PROGRAM Permissives
VAR

	stPermissives			: ST_PermissivesToMainPLC;
	
	AdminFaultBypassOn		: BOOL;
	
	i : INT := 1;
	j : INT := 1;	
END_VAR

//HMI Admin bypass button
AdminFaultBypassOn := HMI_DB.SafetyOK;

//Check to see if any coil is disabled
IF Devices.Coil[1].CoilEnabled = FALSE OR
	Devices.Coil[2].CoilEnabled = FALSE OR
	Devices.Coil[3].CoilEnabled = FALSE OR
	Devices.Coil[4].CoilEnabled = FALSE OR
	Devices.Coil[5].CoilEnabled = FALSE OR
	Devices.Coil[6].CoilEnabled = FALSE OR
	Devices.Coil[7].CoilEnabled = FALSE OR
	Devices.Coil[8].CoilEnabled = FALSE OR
	Devices.Coil[9].CoilEnabled = FALSE OR
	Devices.Coil[10].CoilEnabled = FALSE 
	THEN
		Permissives_DB.AnyCoilDisabled := TRUE;
	ELSE
		Permissives_DB.AnyCoilDisabled := FALSE;
END_IF;

//check to see if each LCP system is ready based on the selected safety parameters.
FOR i := 1 TO 10 BY 1 DO
	IF Devices.Coil[i].AC_Interlock_RlyClose = TRUE AND 
		Devices.Coil[i].ChargeRelay_closed = TRUE AND
		Devices.Coil[i].CoilTemperatureHigh = FALSE AND
		Devices.Coil[i].DumpResistorTemperatureHigh = FALSE AND
		Devices.Coil[i].DumpRelay1_closed = TRUE AND
		Devices.Coil[i].DumpRelay2_closed = TRUE AND
		Devices.Coil[i].FlybackD1_Alive = TRUE AND
		Devices.Coil[i].FlybackD2_Alive = TRUE AND
		Devices.Coil[i].GroundLoopCurrentDetected = FALSE AND
		Devices.Coil[i].Local_StopPB_Pressed = FALSE AND
		Devices.Coil[i].LossPneumaticPressure = FALSE 
		THEN
			Devices.Coil[i].SystemReady := TRUE;
		ELSE
			Devices.Coil[i].SystemReady := FALSE;
	END_IF;
END_FOR;


//Safety Permissives
	//Interlock Safety
	IF (Devices.Coil[1].AC_Interlock_RlyClose = TRUE OR Devices.Coil[1].CoilEnabled = FALSE) AND 
		(Devices.Coil[2].AC_Interlock_RlyClose = TRUE OR Devices.Coil[2].CoilEnabled = FALSE) AND 
		(Devices.Coil[3].AC_Interlock_RlyClose = TRUE OR Devices.Coil[3].CoilEnabled = FALSE) AND
		(Devices.Coil[4].AC_Interlock_RlyClose = TRUE OR Devices.Coil[4].CoilEnabled = FALSE) AND
		(Devices.Coil[5].AC_Interlock_RlyClose = TRUE OR Devices.Coil[5].CoilEnabled = FALSE) AND
		(Devices.Coil[6].AC_Interlock_RlyClose = TRUE OR Devices.Coil[6].CoilEnabled = FALSE) AND
		(Devices.Coil[7].AC_Interlock_RlyClose = TRUE OR Devices.Coil[7].CoilEnabled = FALSE) AND
		(Devices.Coil[8].AC_Interlock_RlyClose = TRUE OR Devices.Coil[8].CoilEnabled = FALSE) AND
		(Devices.Coil[9].AC_Interlock_RlyClose = TRUE OR Devices.Coil[9].CoilEnabled = FALSE) AND 
		(Devices.Coil[10].AC_Interlock_RlyClose = TRUE OR Devices.Coil[10].CoilEnabled = FALSE)
		
		THEN 
			Permissives_DB.AllacInterlock_Closed := TRUE;
		ELSE 
			Permissives_DB.AllacInterlock_Closed := FALSE;
	END_IF;

	//Coil Temperature
	IF Devices.Coil[1].CoilTemperatureHigh = FALSE AND
		Devices.Coil[2].CoilTemperatureHigh = FALSE 
		THEN
			Permissives_DB.All_Coil_TemperatureOK := TRUE;
		ELSE 
			Permissives_DB.All_Coil_TemperatureOK := FALSE;
	END_IF;

	//Dump Resistor Temperature
	IF Devices.Coil[1].DumpResistorTemperatureHigh = FALSE AND
		Devices.Coil[2].DumpResistorTemperatureHigh = FALSE 
		THEN
			Permissives_DB.AllDumpResistorTempOK := TRUE;
		ELSE 
			Permissives_DB.AllDumpResistorTempOK := FALSE;
	END_IF;
	
	//Ground loop current
	IF Devices.Coil[1].GroundLoopCurrentDetected = FALSE AND
		Devices.Coil[2].GroundLoopCurrentDetected = FALSE 
		THEN
			Permissives_DB.NoGroundLoopCurrentDetected := TRUE;
		ELSE 
			Permissives_DB.NoGroundLoopCurrentDetected := FALSE;
	END_IF;
	
	//Flyback Diodes - Not enought time for PI3 - temporarily disabled for PI3
(*	IF ((Devices.coil[1].FlybackD1_Alive = TRUE AND Devices.coil[1].FlybackD2_Alive = TRUE) OR Devices.Coil[1].CoilEnabled = FALSE) AND
		((Devices.coil[2].FlybackD1_Alive = TRUE AND Devices.coil[2].FlybackD2_Alive = TRUE) OR Devices.Coil[2].CoilEnabled = FALSE)
		THEN 
			AllFlybackDiodes_Alive := TRUE;
		ELSE 
			AllFlybackDiodes_Alive := FALSE;
	END_IF;
*)	
	IF (Permissives_DB.All_Coil_TemperatureOK = TRUE AND
		Permissives_DB.AllDumpResistorTempOK = TRUE AND
		Permissives_DB.NoGroundLoopCurrentDetected = TRUE AND
		//AllFlybackDiodes_Alive = TRUE AND 
		Trips_DB.AnyACInterlockFail = FALSE AND
		Trips_DB.AnyHVisoRelayFailed = FALSE AND
		Trips_DB.AnyChargeRlyFail = FALSE AND
		Trips_DB.AnyDumpRlyFail = FALSE AND
		Trips_DB.AnyEstopPressed = FALSE AND
		Permissives_DB.AlldcPSUok = TRUE AND
		MCP_IO.CageEstopCircuitOK = TRUE) OR HMI_DB.SafetyOK = TRUE 
		THEN
			Permissives_DB.SafetyOK := TRUE;
		ELSE 
			Permissives_DB.SafetyOK := FALSE; 
	END_IF;

//Charger Active Status - obsolete
(*
IF (Devices.Coil[1].PSU0_active = TRUE OR Devices.Coil[1].CoilEnabled = FALSE) AND
	(Devices.Coil[2].PSU0_active = TRUE OR Devices.Coil[2].CoilEnabled = FALSE) //AND
	//Coil3.PSU.active AND 
	THEN 
		AllChargers_Active := TRUE;
	ELSE 
		AllChargers_Active := FALSE;
END_IF;
*)

IF (Devices.Coil[1].PSU1_DCOK = TRUE OR Devices.Coil[1].CoilEnabled = FALSE) AND
	(Devices.Coil[2].PSU1_DCOK = TRUE OR Devices.Coil[2].CoilEnabled = FALSE) (*AND Coil3.PSU.active*) AND
	MCP_IO.PSU1_DCOK = TRUE
	THEN 
		Permissives_DB.AlldcPSUok := TRUE;
	ELSE 
		Permissives_DB.AlldcPSUok := FALSE;
END_IF;

//Charger Enabled Status
IF (Devices.Coil[1].ChargerIsEnabled = TRUE OR Devices.Coil[1].CoilEnabled = FALSE) AND
	(Devices.Coil[2].ChargerIsEnabled = TRUE OR Devices.Coil[2].CoilEnabled = FALSE) AND
	(Devices.Coil[3].ChargerIsEnabled = TRUE OR Devices.Coil[3].CoilEnabled = FALSE) AND
	(Devices.Coil[4].ChargerIsEnabled = TRUE OR Devices.Coil[4].CoilEnabled = FALSE) AND
	(Devices.Coil[5].ChargerIsEnabled = TRUE OR Devices.Coil[5].CoilEnabled = FALSE) AND
	(Devices.Coil[6].ChargerIsEnabled = TRUE OR Devices.Coil[6].CoilEnabled = FALSE) AND
	(Devices.Coil[7].ChargerIsEnabled = TRUE OR Devices.Coil[7].CoilEnabled = FALSE) AND	
	(Devices.Coil[8].ChargerIsEnabled = TRUE OR Devices.Coil[8].CoilEnabled = FALSE) AND
	(Devices.Coil[9].ChargerIsEnabled = TRUE OR Devices.Coil[9].CoilEnabled = FALSE) AND
	(Devices.Coil[10].ChargerIsEnabled = TRUE OR Devices.Coil[10].CoilEnabled = FALSE) 
	THEN 
		Permissives_DB.AllChargerEnabled := TRUE;
	ELSE 
		Permissives_DB.AllChargerEnabled := FALSE;
END_IF

//???? need more work
IF ((Devices.Coil[1].chargerSetpoint >= Setpoints.Coil[1].RecipeLocal.chargerSetpoint) OR Devices.Coil[1].CoilEnabled = FALSE) AND
	((Devices.Coil[2].chargerSetpoint >= Setpoints.Coil[2].RecipeLocal.chargerSetpoint) OR Devices.Coil[2].CoilEnabled = FALSE) AND 
	((Devices.Coil[3].chargerSetpoint >= Setpoints.Coil[3].RecipeLocal.chargerSetpoint) OR Devices.Coil[3].CoilEnabled = FALSE) AND
	((Devices.Coil[4].chargerSetpoint >= Setpoints.Coil[4].RecipeLocal.chargerSetpoint) OR Devices.Coil[4].CoilEnabled = FALSE) AND
	((Devices.Coil[5].chargerSetpoint >= Setpoints.Coil[5].RecipeLocal.chargerSetpoint) OR Devices.Coil[5].CoilEnabled = FALSE) AND
	((Devices.Coil[6].chargerSetpoint >= Setpoints.Coil[6].RecipeLocal.chargerSetpoint) OR Devices.Coil[6].CoilEnabled = FALSE) AND
	((Devices.Coil[7].chargerSetpoint >= Setpoints.Coil[7].RecipeLocal.chargerSetpoint) OR Devices.Coil[7].CoilEnabled = FALSE) AND
	((Devices.Coil[8].chargerSetpoint >= Setpoints.Coil[8].RecipeLocal.chargerSetpoint) OR Devices.Coil[8].CoilEnabled = FALSE) AND
	((Devices.Coil[9].chargerSetpoint >= Setpoints.Coil[9].RecipeLocal.chargerSetpoint) OR Devices.Coil[9].CoilEnabled = FALSE) AND
	((Devices.Coil[10].chargerSetpoint >= Setpoints.Coil[10].RecipeLocal.chargerSetpoint) OR Devices.Coil[10].CoilEnabled = FALSE)
	THEN
		GVL.AllChargerReadywithSP := TRUE;
	ELSE
		GVL.AllChargerReadywithSP := FALSE;
END_IF;

//check to see if all cap voltage ready to shoot
FOR i := 1 TO 10 BY 1 DO
		IF ((Devices.Coil[i].CapVoltage[1] >= Devices.Coil[i].chargerSetpoint) AND
			(Devices.Coil[i].CapVoltage[2] >= Devices.Coil[i].chargerSetpoint) AND
			(Devices.Coil[i].CapVoltage[3] >= Devices.Coil[i].chargerSetpoint) AND
			(Devices.Coil[i].CapVoltage[4] >= Devices.Coil[i].chargerSetpoint) AND
			(Devices.Coil[i].CapVoltage[5] >= Devices.Coil[i].chargerSetpoint) AND
			(Devices.Coil[i].CapVoltage[6] >= Devices.Coil[i].chargerSetpoint) AND
			(Devices.Coil[i].CapVoltage[7] >= Devices.Coil[i].chargerSetpoint) AND
			(Devices.Coil[i].CapVoltage[8] >= Devices.Coil[i].chargerSetpoint) AND
			(Devices.Coil[i].CapVoltage[9] >= Devices.Coil[i].chargerSetpoint) AND
			(Devices.Coil[i].CapVoltage[10] >= Devices.Coil[i].chargerSetpoint)) OR 
			Devices.Coil[i].CoilEnabled = FALSE
		THEN
			Devices.Coil[i].AllCapsCharged := TRUE;
	END_IF
END_FOR;
//check to see if all coils are charged
IF Devices.Coil[1].AllCapsCharged = TRUE AND 
	Devices.Coil[2].AllCapsCharged = TRUE AND 
	Devices.Coil[3].AllCapsCharged = TRUE AND 
	Devices.Coil[4].AllCapsCharged = TRUE AND 
	Devices.Coil[5].AllCapsCharged = TRUE AND 
	Devices.Coil[6].AllCapsCharged = TRUE AND 
	Devices.Coil[7].AllCapsCharged = TRUE AND 
	Devices.Coil[8].AllCapsCharged = TRUE AND 
	Devices.Coil[9].AllCapsCharged = TRUE AND 
	Devices.Coil[10].AllCapsCharged = TRUE 
THEN 
	Permissives_DB.AllCoilCapsCharged := TRUE;
ELSE
	Permissives_DB.AllCoilCapsCharged := FALSE;	
END_IF

//check to see if all cap voltage drops to 1
IF ((Devices.Coil[i].CapVoltage[1] <= 1) AND
	(Devices.Coil[i].CapVoltage[2] <= 1) AND
	(Devices.Coil[i].CapVoltage[3] <= 1) AND
	(Devices.Coil[i].CapVoltage[4] <= 1) AND
	(Devices.Coil[i].CapVoltage[5] <= 1) AND
	(Devices.Coil[i].CapVoltage[6] <= 1) AND
	(Devices.Coil[i].CapVoltage[7] <= 1) AND
	(Devices.Coil[i].CapVoltage[8] <= 1) AND
	(Devices.Coil[i].CapVoltage[9] <= 1) AND
	(Devices.Coil[i].CapVoltage[10] <= 1)) OR 
	Devices.Coil[i].CoilEnabled = FALSE
THEN
	Devices.Coil[i].AllCapsCharged := FALSE;
END_IF;



//Charger Relay
IF Devices.Coil[1].ChargeRelay_closed = FALSE AND
	Devices.Coil[2].ChargeRelay_closed = FALSE 
	//coil n
	THEN
		Permissives_DB.AllChargerRelay_Closed := TRUE;
	ELSE 
		Permissives_DB.AllChargerRelay_Closed := FALSE;
END_IF

	
//Dump Relay Status
(* obsolete - use the one at the bottom
IF ((Devices.Coil[1].DumpRelay1_closed = FALSE AND Devices.Coil[1].DumpRelay2_closed = FALSE) OR Devices.Coil[1].CoilEnabled = FALSE) AND
	((Devices.Coil[2].DumpRelay1_closed = FALSE AND Devices.Coil[2].DumpRelay2_closed = FALSE) OR Devices.Coil[2].CoilEnabled = FALSE) AND
	((Devices.Coil[3].DumpRelay1_closed = FALSE AND Devices.Coil[3].DumpRelay2_closed = FALSE) OR Devices.Coil[3].CoilEnabled = FALSE) AND
	((Devices.Coil[4].DumpRelay1_closed = FALSE AND Devices.Coil[4].DumpRelay2_closed = FALSE) OR Devices.Coil[4].CoilEnabled = FALSE) AND
	((Devices.Coil[5].DumpRelay1_closed = FALSE AND Devices.Coil[5].DumpRelay2_closed = FALSE) OR Devices.Coil[5].CoilEnabled = FALSE) AND
	((Devices.Coil[6].DumpRelay1_closed = FALSE AND Devices.Coil[6].DumpRelay2_closed = FALSE) OR Devices.Coil[6].CoilEnabled = FALSE) AND
	((Devices.Coil[7].DumpRelay1_closed = FALSE AND Devices.Coil[7].DumpRelay2_closed = FALSE) OR Devices.Coil[7].CoilEnabled = FALSE) AND
	((Devices.Coil[8].DumpRelay1_closed = FALSE AND Devices.Coil[8].DumpRelay2_closed = FALSE) OR Devices.Coil[8].CoilEnabled = FALSE) AND
	((Devices.Coil[9].DumpRelay1_closed = FALSE AND Devices.Coil[9].DumpRelay2_closed = FALSE) OR Devices.Coil[9].CoilEnabled = FALSE) AND
	((Devices.Coil[10].DumpRelay1_closed = FALSE AND Devices.Coil[10].DumpRelay2_closed = FALSE) OR Devices.Coil[10].CoilEnabled = FALSE)

	THEN
		AllDumpRelayOpen := TRUE;
		ELSE 
			AllDumpRelayOpen := FALSE;
END_IF;
*)	
IF ((Devices.Coil[1].DumpRelay1_closed = TRUE AND Devices.Coil[1].DumpRelay2_closed = TRUE) OR Devices.Coil[1].CoilEnabled = FALSE) AND
	((Devices.Coil[2].DumpRelay1_closed = TRUE AND Devices.Coil[2].DumpRelay2_closed = TRUE) OR Devices.Coil[2].CoilEnabled = FALSE) AND
	((Devices.Coil[3].DumpRelay1_closed = TRUE AND Devices.Coil[3].DumpRelay2_closed = TRUE) OR Devices.Coil[3].CoilEnabled = FALSE) AND
	((Devices.Coil[4].DumpRelay1_closed = TRUE AND Devices.Coil[4].DumpRelay2_closed = TRUE) OR Devices.Coil[4].CoilEnabled = FALSE) AND
	((Devices.Coil[5].DumpRelay1_closed = TRUE AND Devices.Coil[5].DumpRelay2_closed = TRUE) OR Devices.Coil[5].CoilEnabled = FALSE) AND
	((Devices.Coil[6].DumpRelay1_closed = TRUE AND Devices.Coil[6].DumpRelay2_closed = TRUE) OR Devices.Coil[6].CoilEnabled = FALSE) AND
	((Devices.Coil[7].DumpRelay1_closed = TRUE AND Devices.Coil[7].DumpRelay2_closed = TRUE) OR Devices.Coil[7].CoilEnabled = FALSE) AND
	((Devices.Coil[8].DumpRelay1_closed = TRUE AND Devices.Coil[8].DumpRelay2_closed = TRUE) OR Devices.Coil[8].CoilEnabled = FALSE) AND
	((Devices.Coil[9].DumpRelay1_closed = TRUE AND Devices.Coil[9].DumpRelay2_closed = TRUE) OR Devices.Coil[9].CoilEnabled = FALSE) AND
	((Devices.Coil[10].DumpRelay1_closed = TRUE AND Devices.Coil[10].DumpRelay2_closed = TRUE) OR Devices.Coil[10].CoilEnabled = FALSE) 
	THEN
		Permissives_DB.AllDumpRelayOpen := FALSE;
		ELSE
			Permissives_DB.AllDumpRelayOpen := TRUE;;
END_IF;

//any pneumatic pressure loss
FOR i := 1 TO 10 BY 1 DO
	IF Devices.Coil[i].LossPneumaticPressure = FALSE THEN
		Permissives_DB.NoPneumaticPressureLoss := TRUE;
		ELSE 
			Permissives_DB.NoPneumaticPressureLoss := FALSE;
	END_IF
END_FOR

//When disable a coil, ignore the permissives of it
IF Permissives_DB.AnyCoilDisabled = TRUE THEN
	FOR i := 1 TO 10 BY 1 DO
		IF Devices.Coil[i].CoilEnabled = FALSE THEN
			Devices.Coil[i].SystemReady := TRUE;
			Devices.Coil[i].PSU0_active := TRUE;
			Devices.Coil[i].Local_StopPB_Pressed := FALSE;
			Devices.Coil[i].FlybackD1_Alive := TRUE;
			Devices.Coil[i].FlybackD2_Alive := TRUE;
			Devices.Coil[i].DumpResistorTemperatureHigh := FALSE;
			Devices.Coil[i].GroundLoopCurrentDetected := FALSE;
			Devices.Coil[i].CoilTemperatureHigh := FALSE;
			Devices.Coil[i].LossPneumaticPressure := FALSE;
			ELSE
				Devices.Coil[i].SystemReady := FALSE;
		END_IF;
	END_FOR;
END_IF;	


//TURN OFF the outputs of the coil when it is disabled
IF Permissives_DB.AnyCoilDisabled = TRUE THEN
	FOR i := 1 TO 10 BY 1 DO
		IF Devices.Coil[i].CoilEnabled = TRUE THEN
			Devices.Coil[i].CloseACInterlockRly := FALSE;
			Devices.Coil[i].OpenDumpRelays := FALSE;
			Devices.Coil[i].closeChargeRelay := FALSE;
		END_IF;
	END_FOR;
END_IF;

//*******************************************************************//	
//Charge Permissives
IF (Permissives_DB.SafetyOK = TRUE OR HMI_DB.SafetyOK) AND (Permissives_DB.AllDumpRelayOpen = TRUE OR HMI_DB.AllDumpRelaysOpen  = TRUE) AND (Trips_DB.InstrumentationFaulted = FALSE OR HMI_DB.IntrumentationFaulted = FALSE) THEN 
	Permissives_DB.ChargePermOK := TRUE;	
	ELSE Permissives_DB.ChargePermOK := FALSE;	
END_IF;


//Shoot Permissives
IF Permissives_DB.SafetyOK = TRUE AND (Permissives_DB.AlldcPSUok = FALSE OR HMI_DB.AllChargesAreActive = FALSE) AND (Permissives_DB.AllDumpRelayOpen = TRUE OR HMI_DB.AllDumpRelaysOpen = TRUE) THEN
	Permissives_DB.ShootPermOK := TRUE;
	ELSE Permissives_DB.ShootPermOK := FALSE;
END_IF;

//sending permissives to Main PLC (screen room)
stPermissives.All_Coil_TemperatureOK := Permissives_DB.All_Coil_TemperatureOK;
stPermissives.AllacInterlock_Closed := Permissives_DB.AllacInterlock_Closed;
stPermissives.AllChargerEnabled := Permissives_DB.AllChargerEnabled;
stPermissives.AllChargerRelay_Closed := Permissives_DB.AllChargerRelay_Closed;
stPermissives.AlldcPSUok := Permissives_DB.AlldcPSUok;
stPermissives.AllDumpRelayOpen := Permissives_DB.AllDumpRelayOpen;
stPermissives.AllDumpResistorTempOK := Permissives_DB.AllDumpResistorTempOK;
//stPermissives.AllFlybackDiodes_Alive := AllFylbackDiodes_Alive;
stPermissives.AnyCoilDisabled := Permissives_DB.AnyCoilDisabled;
stPermissives.ChargePermOK := Permissives_DB.ChargePermOK;
stPermissives.NoGroundLoopCurrentDetected := Permissives_DB.NoGroundLoopCurrentDetected;
stPermissives.SafetyOK := Permissives_DB.SafetyOK;
stPermissives.ShootPermOK := Permissives_DB.ShootPermOK;
stPermissives.AdminFaultBypassOn := AdminFaultBypassOn;


IF i > 10 THEN
	i := 1;
END_IF;

IF j > 10 THEN
	j := 1;
END_IF;

END_PROGRAM

(* stored: Version 1.1.0.1, ProductVersion 3.1.4024.11
   POU Permissives: Id {10f7449e-ceca-4ebc-9f71-340d6aec6e43}, SpecialFunc None *)
